{attribute 'linkalways'} 
{attribute 'no_explicit_call' := 'This FB is a CLASS and must be accessed using methods or properties'}
{attribute 'enable_dynamic_creation'}
FUNCTION_BLOCK VisionNodePack IMPLEMENTS I_NodePack
VAR
	//node : Node;
END_VAR

METHOD PUBLIC RegisterWithNodeFactory
VAR_INPUT
	NodeFactory : I_NodeFactory;
END_VAR
//NodeFactory.AddNodeAsPrototype('Vision/Node',Node);
END_METHOD

END_FUNCTION_BLOCK

(* stored: Version 1.1.0.1, ProductVersion 3.1.4024.12
   POU VisionNodePack: Id {257fc325-f932-4b89-a50a-e9a0a38418f4}, SpecialFunc None
   Method RegisterWithNodeFactory: Id {9eda346d-cc38-44e9-a636-4948bc24f687} *)
